Staubli VAL3: Prog1.dtx

dio do5 = {link=fiodo5}
public frame fPartReal = {x=0.000, y=0.000, z=0.000, rx=-0.000, ry=0.000, rz=-0.000, fatherId=world[0]}
public jointRx jPark = {j1=0.000, j2=0.000, j3=90.000, j4=0.000, j5=90.000, j6=0.000}
public jointRx jJoint[2]
  [0] = {j1=-0.00000, j2=0.00000, j3=90.00000, j4=0.00000, j5=0.00000, j6=-0.00000}
  [1] = {j1=-8.97077, j2=0.68477, j3=87.65445, j4=79.59684, j5=9.12198, j6=-79.46655}
public mdesc mNomSpeed = {accel=100, vel=100, decel=100, tmax=99999, rmax=99999, blend=off, leave=50, reach=50}
public mdesc mSpeed = {tmax=500.0, rmax=100, leave=0.1, reach=0.1, blend=cartesian}
public num nTraj
num nTimeStop
num nTimeStart
num nMode
num nEtat
public pointRx pPoint[3]
  [0] = {x=885.000, y=-122.343, z=737.831, rx=0.000, ry=90.000, rz=0.000, shoulder=lefty, elbow=epositive, wrist=wpositive, fatherId=fPartReal[0]}
  [1] = {x=966.625, y=-12.231, z=737.831, rx=0.000, ry=90.000, rz=0.000, shoulder=lefty, elbow=epositive, wrist=wpositive, fatherId=fPartReal[0]}
  [2] = {x=881.362, y=96.973, z=737.831, rx=0.000, ry=90.000, rz=0.000, shoulder=lefty, elbow=epositive, wrist=wpositive, fatherId=fPartReal[0]}
public tool tCad = {x=0.000, y=0.000, z=0.000, rx=-0.000, ry=0.000, rz=-0.000, fatherId=flange[0], ioLink=valve1}
